(* CODESYS project Server_01.project

Project tree, tasks and I/O mapping:
  Device : CPX-CEC-C1-V3, Festo AG & Co. KG, order no. 3473128, version 3.5.7.30
      unmapped channels: Rotary switch
    application Application
      libraries: Standard, * (System)
      task MainTask (cyclic, interval t#20ms, priority 20) calls PLC_PRG
      program PLC_PRG [LD]
      Symbols
    PLC_Diagnosis : PLC-Diagnosis, Festo AG & Co. KG, version 3.5.4.1
    CPX_System : CPX_System, Festo AG & Co. KG, order no. 3473128, version 1.233
      CEC_C1_V3 : CEC-C1-V3, Festo AG & Co. KG, order no. 3473128, version 1.233
      _8DI_8DO : 8DI/8DO, Festo AG & Co. KG, order no. 526257, version 1.233
          settings:  = 1;  = 1;  = 1;  = 1;  = 0;  = 1;  = 1;  = 0;  = 0;  = 0;  = 0;  = 0;  = 0;  = 0;  = 0;  = 0;  = 0;  = 0;  = 0;  = 0;  = 0;  = 0;  = 0;  = 0;  = 0;  = 0;  = 0;  = 0;  = 0;  = 0;  = 0;  = 0;  = 0;  = 0;  = 0;  = 0;  = 0;  = 0;  = 0;  = 0;
             = 0;  = 0;  = 0;  = 0;  = 0;  = 0;  = 0;  = 0;  = 0;  = 0;  = 0;  = 0;  = 0;  = 0;  = 0;  = 0;  = 0;  = 0;  = 0;  = 0;  = 0;  = 0;  = 0;  = 0;  = 0;  = 0;  = 0;  = 0;  = 0;  = 0;  = 0;  = 0;  = 0;  = 0;  = 0;  = 0;  = 0;  = 0;  = 0;  = 'PI%i.0.0.1=1';
             = 'PI%i.0.1.1=1';  = 'PI%i.0.2.1=1';  = 'PI%i.1.0.1=1';  = 'PI%i.1.1.1=0';  = 'PI%i.1.4.2=1';  = 'PI%i.1.6.2=1';  = 'PI%i.6.0.1=0';  = 'PI%i.6.1.1=0';  = 'PI%i.6.2.1=0';  = 'PI%i.6.3.1=0';  = 'PI%i.6.4.1=0';  = 'PI%i.6.5.1=0';  = 'PI%i.6.6.1=0';  = 'PI%i.6.7.1=0';  = -;  = -
          input  posicao_atuador_avanco : BOOL  // Input 0.Bit1
          input  posicao_atuador_recuo : BOOL  // Input 0.Bit2
          input  vacuostato : BOOL  // Input 0.Bit3
          input  posicao_rotativo_recuo : BOOL  // Input 0.Bit4
          input  posicao_rotativo_avanco : BOOL  // Input 0.Bit5
          input  peca_armazem : BOOL  // Input 0.Bit6
          output recuo_atuador : BOOL  // Output 0.Bit0
          output vacuo_ventosa : BOOL  // Output 0.Bit1
          output retorno_cilindrico : BOOL  // Output 0.Bit3
          output avanco_cilindrico : BOOL  // Output 0.Bit4
          unmapped channels: Input 0, Output 0
      _8DI_8DO_1 : 8DI/8DO, Festo AG & Co. KG, order no. 526257, version 1.233
          settings:  = 1;  = 1;  = 1;  = 1;  = 0;  = 1;  = 1;  = 0;  = 0;  = 0;  = 0;  = 0;  = 0;  = 0;  = 0;  = 0;  = 0;  = 0;  = 0;  = 0;  = 0;  = 0;  = 0;  = 0;  = 0;  = 0;  = 0;  = 0;  = 0;  = 0;  = 0;  = 0;  = 0;  = 0;  = 0;  = 0;  = 0;  = 0;  = 0;  = 0;
             = 0;  = 0;  = 0;  = 0;  = 0;  = 0;  = 0;  = 0;  = 0;  = 0;  = 0;  = 0;  = 0;  = 0;  = 0;  = 0;  = 0;  = 0;  = 0;  = 0;  = 0;  = 0;  = 0;  = 0;  = 0;  = 0;  = 0;  = 0;  = 0;  = 0;  = 0;  = 0;  = 0;  = 0;  = 0;  = 0;  = 0;  = 0;  = 0;  = 'PI%i.0.0.1=1';
             = 'PI%i.0.1.1=1';  = 'PI%i.0.2.1=1';  = 'PI%i.1.0.1=1';  = 'PI%i.1.1.1=0';  = 'PI%i.1.4.2=1';  = 'PI%i.1.6.2=1';  = 'PI%i.6.0.1=0';  = 'PI%i.6.1.1=0';  = 'PI%i.6.2.1=0';  = 'PI%i.6.3.1=0';  = 'PI%i.6.4.1=0';  = 'PI%i.6.5.1=0';  = 'PI%i.6.6.1=0';  = 'PI%i.6.7.1=0';  = -;  = -
          input  botao_start : BOOL  // Input 0.Bit0
          output led_start : BOOL  // Output 0.Bit0
          unmapped channels: Input 0, Output 0
*)

// Device/Application/PLC_PRG
PROGRAM PLC_PRG
VAR
	posicao_atuador_avancoo:BOOL;
	posicao_atuador_recuoo:BOOL;
	vacuostatoo:BOOL;
	posicao_rotativo_recuoo:BOOL;
	posicao_rotativo_avancoo:BOOL;
	peca_aramzemm:BOOL;
	
	recuo_atuadorr:BOOL;
	vacuo_ventosaa:BOOL;
	retorno_cilindricoo:BOOL;
	avanco_cilindricoo:BOOL;







END_VAR

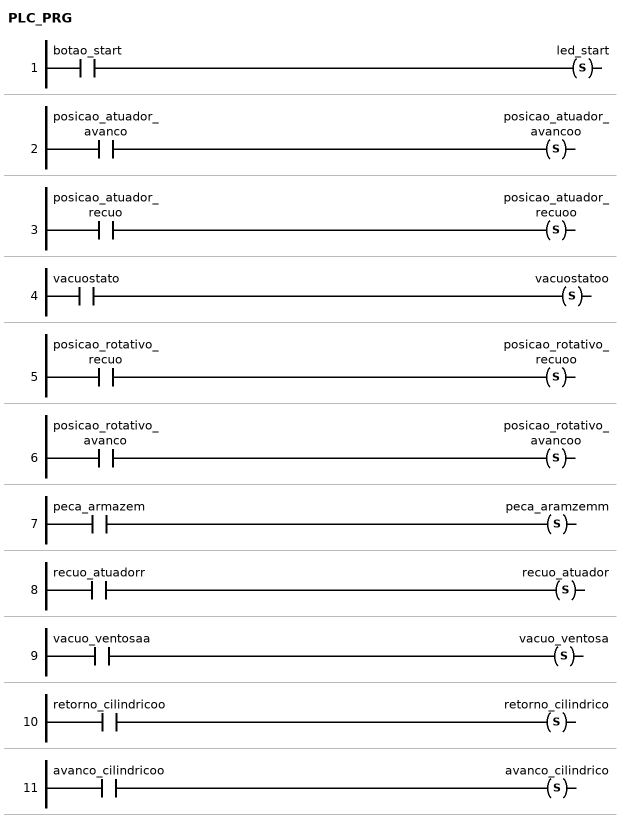
// NETWORK 1
led_start S= botao_start;

// NETWORK 2
posicao_atuador_avancoo S= posicao_atuador_avanco;

// NETWORK 3
posicao_atuador_recuoo S= posicao_atuador_recuo;

// NETWORK 4
vacuostatoo S= vacuostato;

// NETWORK 5
posicao_rotativo_recuoo S= posicao_rotativo_recuo;

// NETWORK 6
posicao_rotativo_avancoo S= posicao_rotativo_avanco;

// NETWORK 7
peca_aramzemm S= peca_armazem;

// NETWORK 8
recuo_atuador S= recuo_atuadorr;

// NETWORK 9
vacuo_ventosa S= vacuo_ventosaa;

// NETWORK 10
retorno_cilindrico S= retorno_cilindricoo;

// NETWORK 11
avanco_cilindrico S= avanco_cilindricoo;

END_PROGRAM
